// TIA Portal project "digital_sensor_app" (V16)

(* hardware
DEVICE "S7-1200 station_1"  S7-1200 Station
   slot 0: "Rack_0"  S7-1200 Rack  Rack  V1.0
   slot 1: "PLC_1"  CPU 1214C DC/DC/Rly  6ES7 214-1HG40-0XB0  V4.4
*)

// ===== PLC "PLC_1"  CPU 1214C DC/DC/Rly =====

VAR_GLOBAL   // PLC tag table "Default tag table"
   "START BUT" AT %I0.0 : Bool;
   "STOP BUT" AT %I0.1 : Bool;
   "SENSÖR 1" AT %I0.2 : Bool;
   "SENSÖR 2" AT %I0.3 : Bool;
   "SENSÖR 3" AT %I0.4 : Bool;
   "PLAT. LİM. SENSÖRÜ" AT %I0.5 : Bool;
   "ASAN. LİM. SENSÖRÜ" AT %I0.6 : Bool;
   "KONVEYÖR 1" AT %Q0.0 : Bool;
   "KONVEYÖR 2" AT %Q0.1 : Bool;
   "PLAT. İLERİ. HAR." AT %Q0.2 : Bool;
   "PLAT. DÖNDÜR" AT %Q0.3 : Bool;
   "ASAN. İLERİ" AT %Q0.4 : Bool;
   "ASAN. YUKARI" AT %Q0.5 : Bool;
   "PLAT. DÖN. SENSÖRÜ" AT %I0.7 : Bool;
END_VAR

// folder: System blocks/Program resources

DATA_BLOCK "TIMER 1"   // DB1
{ S7_Optimized_Access := 'TRUE' }
AUTHOR : Simatic
FAMILY : IEC
NAME : IEC_TMR
VERSION : 1.0
// stored: InstanceOfName IEC_TIMER
"IEC_TIMER"
BEGIN
END_DATA_BLOCK

// folder: (top level)

ORGANIZATION_BLOCK "Main"   // OB1, LAD, ProgramCycle
TITLE = "Main Program Sweep (Cycle)"
{ S7_Optimized_Access := 'TRUE' }
VERSION : 0.1
   VAR_INPUT
      Initial_Call : Bool;   // Initial call of this OB
      Remanence : Bool;   // =True, if remanent data are available
   END_VAR
BEGIN

REGION Network 1
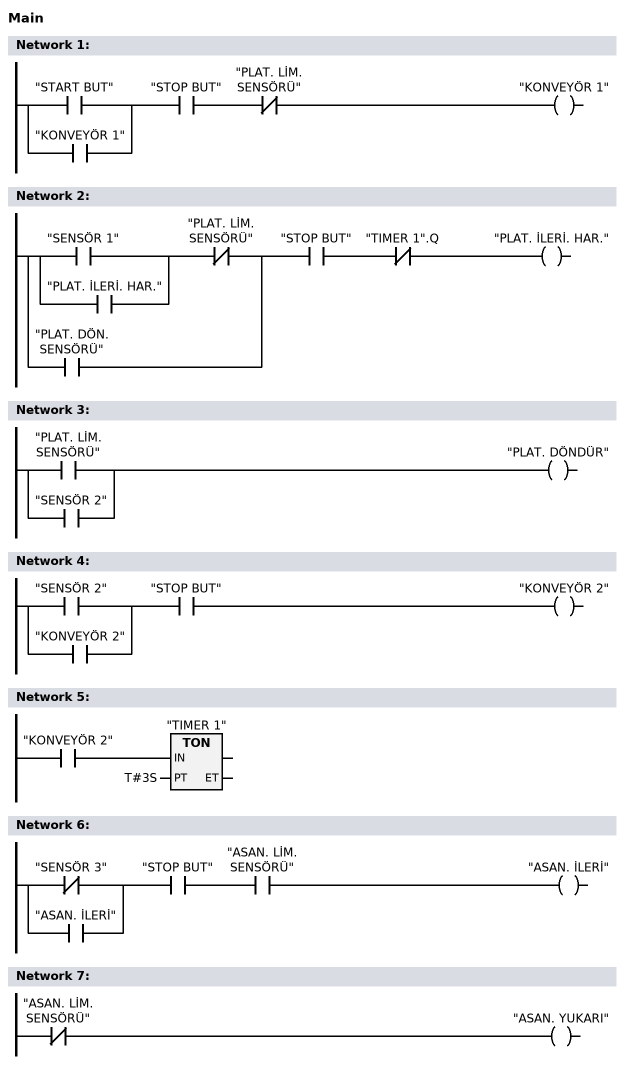
   RUNG wire#powerrail
      Contact( "START BUT" )
      wire#w1
      Contact( "STOP BUT" )
      I_Contact( "PLAT. LİM. SENSÖRÜ" )
      Coil( "KONVEYÖR 1" )
   END_RUNG
   RUNG wire#powerrail
      Contact( "KONVEYÖR 1" )
   END_RUNG wire#w1
   // the same network as SCL:
   "KONVEYÖR 1" := ("START BUT" OR "KONVEYÖR 1") AND "STOP BUT" AND NOT "PLAT. LİM. SENSÖRÜ";
END_REGION

REGION Network 2
   RUNG wire#powerrail
      Contact( "SENSÖR 1" )
      wire#w1
      I_Contact( "PLAT. LİM. SENSÖRÜ" )
      wire#w2
      Contact( "STOP BUT" )
      I_Contact( "TIMER 1".Q )
      Coil( "PLAT. İLERİ. HAR." )
   END_RUNG
   RUNG wire#powerrail
      Contact( "PLAT. İLERİ. HAR." )
   END_RUNG wire#w1
   RUNG wire#powerrail
      Contact( "PLAT. DÖN. SENSÖRÜ" )
   END_RUNG wire#w2
   // the same network as SCL:
   "PLAT. İLERİ. HAR." := ((("SENSÖR 1" OR "PLAT. İLERİ. HAR.") AND NOT "PLAT. LİM. SENSÖRÜ") OR "PLAT. DÖN. SENSÖRÜ") AND "STOP BUT" AND NOT "TIMER 1".Q;
END_REGION

REGION Network 3
   RUNG wire#powerrail
      Contact( "PLAT. LİM. SENSÖRÜ" )
      wire#w1
      Coil( "PLAT. DÖNDÜR" )
   END_RUNG
   RUNG wire#powerrail
      Contact( "SENSÖR 2" )
   END_RUNG wire#w1
   // the same network as SCL:
   "PLAT. DÖNDÜR" := "PLAT. LİM. SENSÖRÜ" OR "SENSÖR 2";
END_REGION

REGION Network 4
   RUNG wire#powerrail
      Contact( "SENSÖR 2" )
      wire#w1
      Contact( "STOP BUT" )
      Coil( "KONVEYÖR 2" )
   END_RUNG
   RUNG wire#powerrail
      Contact( "KONVEYÖR 2" )
   END_RUNG wire#w1
   // the same network as SCL:
   "KONVEYÖR 2" := ("SENSÖR 2" OR "KONVEYÖR 2") AND "STOP BUT";
END_REGION

REGION Network 5
   "TIMER 1".TON(IN := "KONVEYÖR 2", PT := T#3S);
END_REGION

REGION Network 6
   RUNG wire#powerrail
      I_Contact( "SENSÖR 3" )
      wire#w1
      Contact( "STOP BUT" )
      Contact( "ASAN. LİM. SENSÖRÜ" )
      Coil( "ASAN. İLERİ" )
   END_RUNG
   RUNG wire#powerrail
      Contact( "ASAN. İLERİ" )
   END_RUNG wire#w1
   // the same network as SCL:
   "ASAN. İLERİ" := (NOT "SENSÖR 3" OR "ASAN. İLERİ") AND "STOP BUT" AND "ASAN. LİM. SENSÖRÜ";
END_REGION

REGION Network 7
   RUNG wire#powerrail
      I_Contact( "ASAN. LİM. SENSÖRÜ" )
      Coil( "ASAN. YUKARI" )
   END_RUNG
   // the same network as SCL:
   "ASAN. YUKARI" := NOT "ASAN. LİM. SENSÖRÜ";
END_REGION
END_ORGANIZATION_BLOCK